INTERFACE I_BitDatatype EXTENDS I_Datatype

PROPERTY PUBLIC BitOffset : DWORD
GET
END_GET
END_PROPERTY

PROPERTY PUBLIC ByteOffset : PVOID
GET
END_GET
END_PROPERTY

PROPERTY PUBLIC Parent : I_StructuredDatatype
GET
END_GET
END_PROPERTY

PROPERTY PUBLIC Value : BOOL
GET
END_GET
SET
END_SET
END_PROPERTY

END_INTERFACE

(* stored: Version 1.1.0.1, ProductVersion 3.1.4024.12
   Itf I_BitDatatype: Id {2480a7fa-6764-4cb3-a79d-bb0b9c7ea0b4}
   Property BitOffset: Id {6125247b-9187-4db4-b9f9-a648aee1ef87}
   Get Get: Id {8b3c4109-448b-4b27-89f5-50b4b3c0b13d}
   Property ByteOffset: Id {57a625af-72e1-4fe7-abe3-71dd2c1cf834}
   Get Get: Id {580f1acf-53de-4490-a3ef-2fdc68e095df}
   Property Parent: Id {5005ac07-e597-4545-aabc-7c29501ee657}
   Get Get: Id {5f0edae0-8fe9-403a-bb62-6df48ca4b9a7}
   Property Value: Id {1632a37e-4c6a-4f6b-9f27-b63ea473aa18}
   Get Get: Id {2efd7fc3-cf8c-4dda-8a0a-a14f28756314}
   Set Set: Id {5dd27865-d937-40f3-ba53-28a1278fd75b} *)
